Fanuc KAREL source: kt00506.KL

-- PROVISIONAL review KL for V940-1; original PC SHA256 2a9f0d998175b71723c91c043fbdf7345a00203c8611ed264ee6505796749901
-- Incomplete behavior may be omitted. Consult companion uncertainty JSON. Do not deploy.
PROGRAM KT00506
%NOLOCKGROUP
-- UNRESOLVED_DECL P1 type=000102
-- UNRESOLVED_DECL P2 type=000106
-- UNRESOLVED_DECL OUT type=000106
BEGIN
  -- V9_ZERO_TABLE_METADATA_HINT layout=0001; no indexed target words; source/name/runtime held
  -- UNRESOLVED_PC offsets 5-20; opcodes 2E,22,32,35
  -- UNRESOLVED_PC offsets 25-40; opcodes 2E,22,32,35
  -- UNRESOLVED_PC offsets 45-84; opcodes 49,7E,49,7E,60,7E,4A
  -- UNRESOLVED_PC offsets 89-93; opcodes 7F
END KT00506
